// SIMATIC S7-200 project (STEP 7-Micro/WIN), CPU 221 REL 01.10

ORGANIZATION_BLOCK PRINCIPAL:OB1
TITLE=MOOESTABLE CON RESET AUTOMÁTICO  /  JEVG
BEGIN
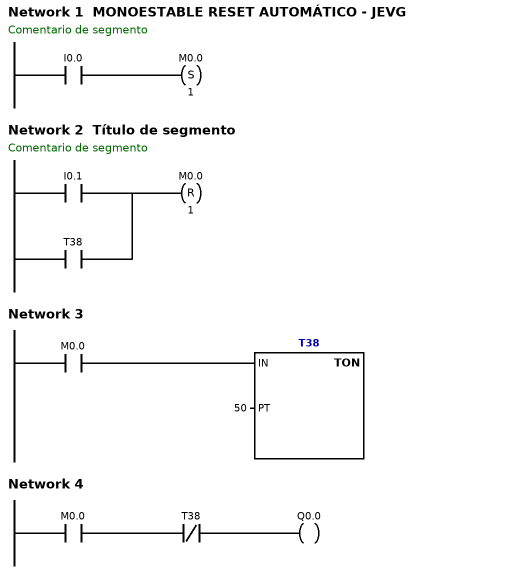
Network 1 // MONOESTABLE RESET AUTOMÁTICO - JEVG
// Comentario de segmento
LD     I0.0
S      M0.0, 1
Network 2 // Título de segmento
// Comentario de segmento
LD     I0.1
O      T38
R      M0.0, 1
Network 3
LD     M0.0
TON    T38, 50
Network 4
LD     M0.0
AN     T38
=      Q0.0
END_ORGANIZATION_BLOCK
